FUNCTION CheckNotOk : BOOL
VAR_INPUT
	hr : HRESULT;
END_VAR

CheckNotOk := (hr <> S_OK);

END_FUNCTION

(* stored: Version 1.1.0.1, ProductVersion 3.1.4024.11
   POU CheckNotOk: Id {3eb1a9bb-8d6a-407a-8ada-d3d1d030b038}, SpecialFunc None *)
